// TIA Portal project "SDRIVE" (V17)

(* hardware
DEVICE "HMI_1"  TP700 Comfort
   slot 0: "HMI_1"  TP700 Comfort  6AV2 124-0GC01-0AX0  15.0.0.0
   slot 1: "HMI_RT_1"  TP700 Comfort  6AV2 124-0GC01-0AX0  15.0.0.0
   slot 5: "HMI_1.IE_CP_1"  PROFINET Interface  15.0.0.0
      slot 1: "PROFINET Interface_1"  PROFINET Interface
         slot 1: "Port_1"  Port
         slot 2: "Port_2"  Port
   slot 7: "HMI_1.MPI/DP_CP_1"  MPI/DP Interface  15.0.0.0
DEVICE "S7-1200 station_1"  S7-1200 Station
   slot 0: "Rack_0"  S7-1200 Rack  Rack  V1.0
   slot 1: "PLC_1"  CPU 1214C DC/DC/DC  6ES7 214-1AG40-0XB0  V4.0
*)

// ===== PLC "PLC_1"  CPU 1214C DC/DC/DC =====

ORGANIZATION_BLOCK "Main"   // OB1, LAD, ProgramCycle
TITLE = "Main Program Sweep (Cycle)"
{ S7_Optimized_Access := 'TRUE' }
VERSION : 0.1
   VAR_INPUT
      Initial_Call : Bool;   // Initial call of this OB
      Remanence : Bool;   // =True, if remanent data are available
   END_VAR
BEGIN
END_ORGANIZATION_BLOCK

(* ===== HMI "HMI_RT_1" =====
system functions are stored by id; their names below are inferred from use
connection "HMI_Connection_1": ETHERNET, S7_1200_OMS

HMI tags "Default tag table"
   "Tag_ScreenNumber" : UInt, internal

screen "Root screen" 800x420, template "Template_1"
   on GenerateScreen: SetTag("Tag_ScreenNumber", 1)
   TextField "HmiScreenItemData_1" at 151,166 size 576x25; Text 'Welcome to HMI_1 (TP700 Comfort)!'
   Button "HmiScreenItemData" at 115,36 size 159x47; TextOff 'Screen0'; PictureOff "Navigates to Screen0 for TP700 Comfort 15.0.0.0"; PictureOn "Navigates to Screen0 for TP700 Comfort 15.0.0.0"
      on Release: ActivateScreen("Screen0", 0)

Template "Template_1" 800x420
   Button "Alarms" at 1,2 size 78x58; TextOff 'Alarms'; PictureOff "AlarmDisplay_TP700_Comfort_TR"; PictureOn "AlarmDisplay_TP700_Comfort_TR"
      on Release: function_ef3f5d25("Alarm window_Unacknowledged", -1)
   Button "Template_Button" at 1,62 size 78x58; TextOff 'Text'
   Button "Template_Button_1" at 1,121 size 78x58; TextOff 'Text'
   Button "Template_Button_2" at 1,181 size 78x58; TextOff 'Text'
   Button "Template_Button_3" at 1,241 size 78x58; TextOff 'Text'
   Button "Template_Button_4" at 1,301 size 78x58; TextOff 'Text'
   Button "Template_Button_5" at 720,360 size 78x58; TextOff 'Text'
   Button "Template_Button_6" at 640,360 size 78x58; TextOff 'Text'
   Button "Template_Button_7" at 560,360 size 78x58; TextOff 'Text'
   Button "Template_Button_8" at 480,360 size 78x58; TextOff 'Text'
   Button "Template_Button_9" at 400,360 size 78x58; TextOff 'Text'
   Button "Template_Button_10" at 321,360 size 78x58; TextOff 'Text'
   Button "Template_Button_11" at 241,360 size 78x58; TextOff 'Text'
   Button "Template_Button_12" at 161,360 size 78x58; TextOff 'Text'
   Button "Template_Button_13" at 81,360 size 78x58; TextOff 'Text'
   Button "Template_Button_14" at 1,360 size 78x58; TextOff 'Text'

screen "Screen0" 800x420, template "Template_1"
   on GenerateScreen: SetTag("Tag_ScreenNumber", 2)
   TextField "HmiScreenItemData" at 151,166 size 576x25; Text 'Screen0'
   Button "Back" at 80,1 size 159x47; TextOff 'Back'
      on Release: ActivateScreen("Root screen", 0)
*)